(*
SPDX-FileCopyrightText: Â© 2026 Oleksandr Tiutyk <trofimich@gmail.com>
SPDX-License-Identifier: MIT
License: https://opensource.org/license/mit
*)

(*!
<summary>Policy that sets parent error but continues cyclic execution.</summary>
<description>
Returns CHILD_CRITICAL_ERROR_REACTION.SET_ERROR_AND_CONTINUE when a child component fails.
</description>
*)

{attribute 'no_explicit_call' := 'do not call this function block directly'}
FUNCTION_BLOCK SetErrorAndContinueAfterChildCriticalErrorHandlingPolicy EXTENDS TOF_Core.Object IMPLEMENTS IChildCriticalErrorHandlingPolicy
VAR_STAT
	{attribute 'hide'} 
	_ClassName : STRING := __POUNAME();
END_VAR

(*!
<summary>Gets the class name of the policy.</summary>
*)
{attribute 'monitoring' := 'call'}
PROPERTY ClassName : REFERENCE TO STRING
GET
ClassName REF= _ClassName;
END_GET
END_PROPERTY

(*!
<summary>Returns CHILD_CRITICAL_ERROR_REACTION.SET_ERROR_AND_CONTINUE for the child error.</summary>
<param name="childWithError">Child component that reported the error.</param>
<param name="handlingObject">Parent component handling the failure.</param>
*)
METHOD HandleChildCriticalError : CHILD_CRITICAL_ERROR_REACTION
VAR_INPUT
	childWithError : IChildAutomationComponent;
	handlingObject : TOF_Core.IObject;
END_VAR
HandleChildCriticalError := CHILD_CRITICAL_ERROR_REACTION.SET_ERROR_AND_CONTINUE;
END_METHOD

(*!
<summary>Gets the namespace of the policy.</summary>
*)
{attribute 'monitoring' := 'call'}
PROPERTY NamespaceName : REFERENCE TO STRING
GET
NamespaceName REF= CurrentNamespace.Name;
END_GET
END_PROPERTY

(*!
<summary>Gets instance memory footprint in bytes.</summary>
*)
{attribute 'monitoring' := 'call'}
PROPERTY SelfSize : ULINT
GET
SelfSize := XSIZEOF(THIS^);
END_GET
END_PROPERTY

END_FUNCTION_BLOCK

(* stored: Version 1.1.0.1
   POU SetErrorAndContinueAfterChildCriticalErrorHandlingPolicy: Id {931907ff-f865-432f-ab0d-7f9f25bff484}, SpecialFunc None
   Property ClassName: Id {b5c5ec87-7113-42c9-a9b1-fcaab1bf4332}
   Get Get: Id {117bd844-8c89-46cf-87f8-a048ccab2400}
   Method HandleChildCriticalError: Id {57b6ea3c-6704-4243-9d3c-afa36e5e0362}
   Property NamespaceName: Id {d3613df1-4666-45c8-bc96-384d41ebf4c5}
   Get Get: Id {db0cd3c5-d174-4e3e-b485-493f2b6711d0}
   Property SelfSize: Id {3c5b3a4a-0df8-4e23-9ced-915e97489dd3}
   Get Get: Id {ffe7c504-c6a6-4356-9587-6e2bc32017ca} *)
